{attribute 'qualified_only'}
VAR_GLOBAL
	


END_VAR

(* stored: Version 1.1.0.1
   GVL GVL_Params: Id {bf8b644f-3abc-0bdd-3922-9080e24117e1} *)
